FUNCTION_BLOCK AdsWriteVariable
VAR_INPUT
	NetID: STRING := '';
	Name: STRING;
	EN: BOOL;
	Source: PVOID;
END_VAR
VAR_OUTPUT
	ENO: BOOL;
END_VAR
VAR
	PLC_ReadSymInfoByName: PLC_ReadSymInfoByName;
	ADSWRITE: ADSWRITE;
	State : INT := 0;
END_VAR

CASE State OF
0:
	IF EN THEN
		State := 1;
	END_IF
1:	
	PLC_ReadSymInfoByName(
		NETID := NetID, 
		PORT := 851, 
		SYMNAME := Name,
		TMOUT := T#5S,
		START := TRUE
	);
	State := 2;
2:
	PLC_ReadSymInfoByName();
	IF NOT PLC_ReadSymInfoByName.BUSY THEN
		PLC_ReadSymInfoByName(START := FALSE);
		ADSWRITE(
			NETID:= '',
			PORT:= 851,
			IDXGRP:= PLC_ReadSymInfoByName.SYMINFO.idxGroup,
			IDXOFFS:= PLC_ReadSymInfoByName.SYMINFO.idxOffset,
			LEN:= SIZEOF(PLC_ReadSymInfoByName.SYMINFO.byteSize),
			SRCADDR:= Source,
			WRITE:= TRUE,
			TMOUT:= T#5S,
		);
		State := 3;		
	END_IF
	IF NOT EN THEN
		ADSWRITE(WRITE := FALSE);
		ENO := FALSE;
		State := 0;
	END_IF
3:
	ADSWRITE();
	IF NOT ADSWRITE.BUSY THEN
		ENO := TRUE;
		ADSWRITE(WRITE := FALSE);
	END_IF
	IF NOT EN THEN
		ADSWRITE(WRITE := FALSE);
		ENO := FALSE;
		State := 0;
	END_IF
END_CASE

END_FUNCTION_BLOCK

(* stored: Version 1.1.0.1, ProductVersion 3.1.4024.6
   POU AdsWriteVariable: Id {0bb084a0-59da-462e-b6e8-e1ae0d184846}, SpecialFunc None *)
